Fanuc KAREL source: kt00016.KL

-- PROVISIONAL review KL for V770-1; original PC SHA256 7322265496b2264981220a96c93a25ccb373ed21a37217ba993c79032235504f
-- Incomplete behavior may be omitted. Consult companion uncertainty JSON. Do not deploy.
PROGRAM KT00016
%NOLOCKGROUP
VAR
  R1 : REAL
  OUT : REAL
-- UNRESOLVED_DECL H2 type=002017
BEGIN
  -- UNRESOLVED_PC offsets 5-16; opcodes 2E,23
  -- UNRESOLVED_PC offsets 21-35; opcodes 2E,22,9D,33,B4
  -- UNRESOLVED_PC offsets 40-63; opcodes 21,22,9D,33,B3,64,69,23
  -- UNRESOLVED_PC offsets 68-72; opcodes 7F
END KT00016
